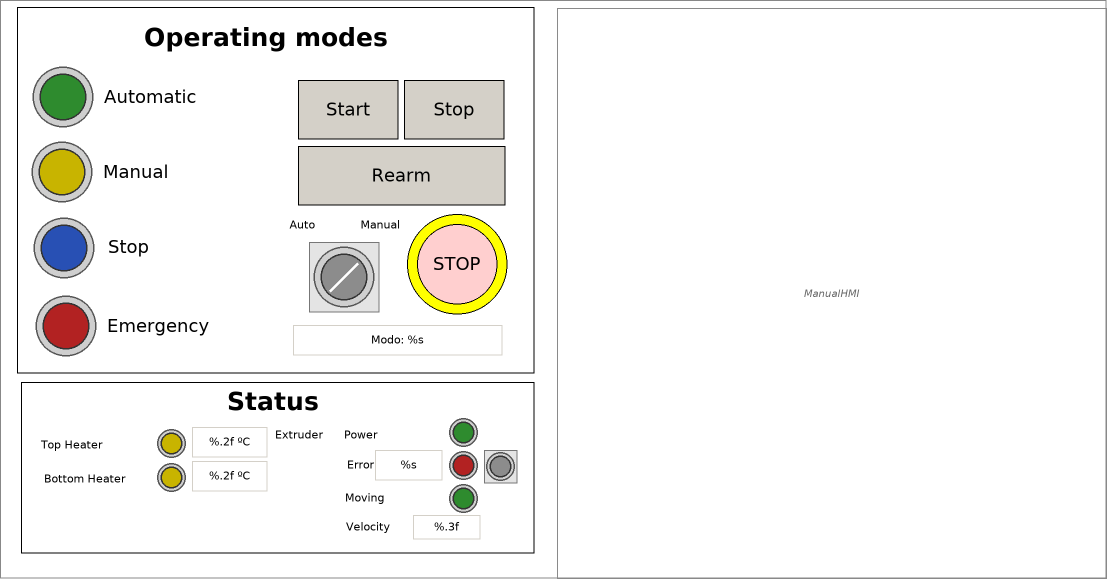
VISUALIZATION MainHMI  // 1107x579
    RoundedRectangle (21,382 513x171)
    RoundedRectangle (17,7 517x366)
    Lamp1 (28,62 70x70), variable: VisuLogic.L_Run, style: Lamp-Lamp1-Green
    Label (101,82 118x30), "Automatic"
    Label (100,157 119x30), "Manual"
    Lamp1 (27,137 70x70), variable: VisuLogic.L_Manual, style: Lamp-Lamp1-Yellow
    Label (105,232 114x30), "Stop"
    Lamp1 (29,213 70x70), variable: VisuLogic.L_StopOP, style: Lamp-Lamp1-Blue
    Label (104,311 115x30), "Emergency"
    Lamp1 (31,291 70x70), variable: VisuLogic.L_StopEM, style: Lamp-Lamp1-Red
    Rectangle (298,80 100x59), "Start"
        tap HMI.Bt_Run
    Rectangle (404,80 100x59), "Stop"
        tap HMI.Bt_Stop
    Rectangle (298,146 207x59), "Rearm"
        tap HMI.Bt_Rearm
    Ellipse (407,214 100x100)
    Ellipse (417,224 80x80), "STOP"
        toggle HMI.Bt_EmStop
    RotarySwitch (309,242 70x70), variable: HMI.S_ManAuto, behaviour: TOGGLE, style: Switch-RotarySwitch-Gray
    Label (284,210 122x30), "Auto Manual"
    Label (124,22 284x30), "Operating modes"
    Label (131,386 284x30), "Status"
    Lamp1 (155,427 33x33), variable: IO.Q_HeaterT, style: Lamp-Lamp1-Yellow
    Lamp1 (155,461 33x33), variable: IO.Q_HeaterB, style: Lamp-Lamp1-Yellow
    Label (38,430 150x30), "Top Heater"
    Label (41,464 150x30), "Bottom Heater"
    Textfield (192,427 75x30), "%.2f ºC", text variable: GVL.TempTerT
    Textfield (192,461 75x30), "%.2f ºC", text variable: GVL.TempTerB
    Label (272,420 57x30), "Extruder"
    Lamp1 (447,449 33x33), variable: MC.Extruder.Status.Error, style: Lamp-Lamp1-Red
    Lamp1 (447,416 33x33), variable: Motion.FB_Power.Status, style: Lamp-Lamp1-Green
    Label (341,420 57x30), "Power"
    Label (344,450 57x30), "Error"
    Textfield (375,450 67x30), "%s", text variable: MC.Extruder.Status.ErrorID
    Lamp1 (447,482 33x33), variable: MC.Extruder.Status.Moving, style: Lamp-Lamp1-Green
    Label (342,483 103x30), "Moving"
    Label (343,512 57x30), "Velocity"
    Textfield (413,515 67x24), "%.3f", text variable: MC.Extruder.NcToPlc.ActVelo
    Textfield (293,325 209x30), "Modo: %s", text variable: GVL.Mode
    PushSwitch (484,450 33x33), variable: HMI.Bt_ResetAxis, behaviour: TAP, style: Switch-PushSwitch-Gray
    TabControl (557,8 550x571)
        shows ManualHMI()
        shows VisionHMI()
        shows BasicHMI()
        [0]: TabTitle=Manual
        [1]: TabTitle=Camera
        [2]: TabTitle=Basic Mode
END_VISUALIZATION

(* stored: Version 1.1.0.1, ProductVersion 3.1.4024.9
   Visu MainHMI: Id {0172a1fd-df4d-437d-8e15-edc9aa511a18} *)
